FUNCTION TFCylinder_HasCommand : bool
VAR_INPUT
	Command: CylinderCommand;
END_VAR
VAR
END_VAR

Cylinder_HasCommand:=
Command.Deactivation OR 
Command.Activation OR 
Command.Hold OR
Command.Abort;

END_FUNCTION

(* stored: Version 1.1.0.1, ProductVersion 3.1.4024.11
   POU TFCylinder_HasCommand: Id {29c6a6de-24ef-44f0-8107-5d892edb72e5}, SpecialFunc None *)
